{attribute 'qualified_only'}
{attribute 'strict'}
TYPE HomingMode :
(
	Default := MC_DefaultHoming,
	Direct := MC_Direct,
	ForceCalibration := MC_ForceCalibration,
	ResetCalibration := MC_ResetCalibration
) INT;
END_TYPE

(* stored: Version 1.1.0.1, ProductVersion 3.1.4024.12
   DUT HomingMode: Id {bca107ba-ce78-0940-1235-c7d99777d92a} *)
